Staubli VAL3: dioItem.dtx

public bool bActive
public string sID
public string sName
public dio dDio
public bool bEnable
